// TIA Portal V20 export
// export: Created 2026-04-11T06:02:29.9652501Z, ExportSetting WithDefaults, DisplayName Totally Integrated Automation Portal, DisplayVersion V20, DisplayName TIA Portal Openness, DisplayVersion V20, DisplayName TIA Portal Version Control Interface, DisplayVersion V20, DisplayName STEP 7 Professional, DisplayVersion V20, DisplayName STEP 7 Safety, DisplayVersion V20, DisplayName WinCC Basic/Comfort/Advanced, DisplayVersion V20, DisplayName WinCC Unified, DisplayVersion V20
TYPE "udtError_Motor"
// stored: IsFailsafeCompliant false
   STRUCT
      MotorProtectorTripped { ExternalWritable := 'False'} : Bool;   // Motor protector tripped
      LocalDisconnectOff { ExternalWritable := 'False'} : Bool;   // Local disconnect off
      ClutchTripped { ExternalWritable := 'False'} : Bool;   // Clutch tripped
      NoSignalForward { ExternalWritable := 'False'} : Bool;   // No signal from forward contactor
      NoSignalReverse { ExternalWritable := 'False'} : Bool;   // No signal from Reverse contactor
      MotorNotStopped { ExternalWritable := 'False'} : Bool;   // Motor doesn't stop
   END_STRUCT;
END_TYPE
